// TIA Portal project "Project1" (V15.1)

(* hardware
DEVICE "S7-1200 station_1"  S7-1200 Station
   slot 0: "Rack_0"  S7-1200 Rack  Rack  V1.0
   slot 1: "PLC_1"  CPU 1214C AC/DC/Rly  6ES7 214-1BG40-0XB0  V4.2
DEVICE "HMI_1"  KTP700 Basic PN
   slot 0: "HMI_1"  KTP700 Basic PN  6AV2 123-2GB03-0AX0  15.1.0.0
   slot 1: "HMI_RT_1"  KTP700 Basic PN  6AV2 123-2GB03-0AX0  15.1.0.0
   slot 5: "HMI_1.IE_CP_1"  PROFINET Interface  15.0.1.0
      slot 1: "Interface PROFINET_1"  PROFINET Interface
         slot 1: "Port_1"  Port
*)

// ===== PLC "PLC_1"  CPU 1214C AC/DC/Rly =====

VAR_GLOBAL   // PLC tag table "Default tag table"
   "AU" AT %I0.0 : Bool;
   "X0" AT %M0.1 : Bool;
   "X30" AT %M0.2 : Bool;
   "Auto" AT %I0.3 : Bool;
   "Manuel" AT %I0.4 : Bool;
   "X31" AT %M0.5 : Bool;
   "X32" AT %M0.6 : Bool;
   "X20" AT %M0.7 : Bool;
   "BP1" AT %I1.0 : Bool;
   "BP2" AT %I1.2 : Bool;
   "X21" AT %M1.2 : Bool;
   "X22" AT %M1.4 : Bool;
   "CV1" AT %Q1.4 : Bool;
   "CV2" AT %Q1.6 : Bool;
   "NB1" AT %I1.6 : Bool;
   "NB2" AT %I1.7 : Bool;
   "X1" AT %M2.0 : Bool;
   "X2" AT %M2.1 : Bool;
   "X3" AT %M2.2 : Bool;
   "X4" AT %M2.3 : Bool;
   "X5" AT %M2.4 : Bool;
   "NH1" AT %I0.5 : Bool;
   "NH2" AT %I0.6 : Bool;
   "X10" AT %M2.7 : Bool;
   "X11" AT %M3.0 : Bool;
END_VAR

FUNCTION "GC" : Void   // FC1, LAD
{ S7_Optimized_Access := 'TRUE' }
VERSION : 0.1
BEGIN

REGION Network 1
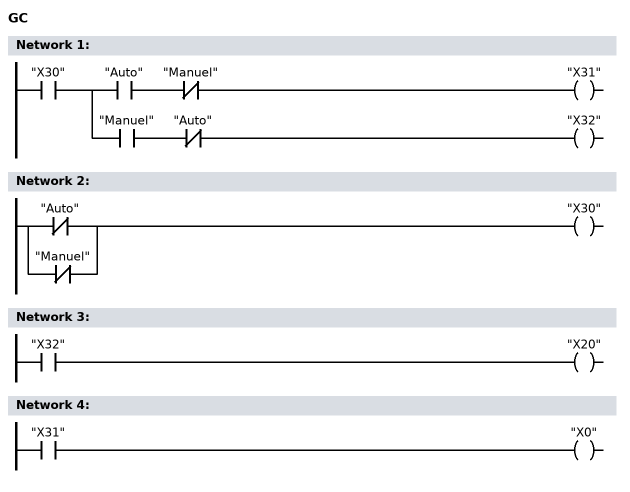
   RUNG wire#powerrail
      Contact( "X30" )
      wire#w1
      Contact( "Auto" )
      I_Contact( "Manuel" )
      Coil( "X31" )
   END_RUNG
   RUNG wire#w1
      Contact( "Manuel" )
      I_Contact( "Auto" )
      Coil( "X32" )
   END_RUNG
   // the same network as SCL:
   "X31" := "X30" AND "Auto" AND NOT "Manuel";
   "X32" := "X30" AND "Manuel" AND NOT "Auto";
END_REGION

REGION Network 2
   RUNG wire#powerrail
      I_Contact( "Auto" )
      wire#w1
      Coil( "X30" )
   END_RUNG
   RUNG wire#powerrail
      I_Contact( "Manuel" )
   END_RUNG wire#w1
   // the same network as SCL:
   "X30" := NOT "Auto" OR NOT "Manuel";
END_REGION

REGION Network 3
   RUNG wire#powerrail
      Contact( "X32" )
      Coil( "X20" )
   END_RUNG
   // the same network as SCL:
   "X20" := "X32";
END_REGION

REGION Network 4
   RUNG wire#powerrail
      Contact( "X31" )
      Coil( "X0" )
   END_RUNG
   // the same network as SCL:
   "X0" := "X31";
END_REGION
END_FUNCTION

FUNCTION "GMM" : Void   // FC2, LAD
{ S7_Optimized_Access := 'TRUE' }
VERSION : 0.1
   VAR_TEMP   // added for the SCL form of the ladder/FBD networks
      _w1 : Bool;
   END_VAR
BEGIN

REGION Network 1
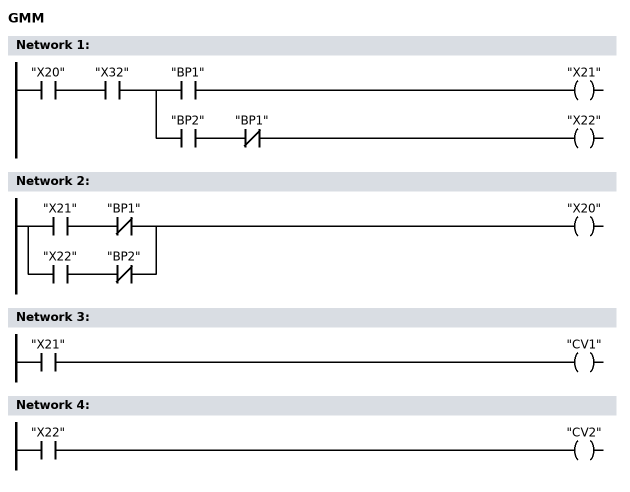
   RUNG wire#powerrail
      Contact( "X20" )
      Contact( "X32" )
      wire#w1
      Contact( "BP1" )
      Coil( "X21" )
   END_RUNG
   RUNG wire#w1
      Contact( "BP2" )
      I_Contact( "BP1" )
      Coil( "X22" )
   END_RUNG
   // the same network as SCL:
   #_w1 := "X20" AND "X32";
   "X21" := #_w1 AND "BP1";
   "X22" := #_w1 AND "BP2" AND NOT "BP1";
END_REGION

REGION Network 2
   RUNG wire#powerrail
      Contact( "X21" )
      I_Contact( "BP1" )
      wire#w1
      Coil( "X20" )
   END_RUNG
   RUNG wire#powerrail
      Contact( "X22" )
      I_Contact( "BP2" )
   END_RUNG wire#w1
   // the same network as SCL:
   "X20" := ("X21" AND NOT "BP1") OR ("X22" AND NOT "BP2");
END_REGION

REGION Network 3
   RUNG wire#powerrail
      Contact( "X21" )
      Coil( "CV1" )
   END_RUNG
   // the same network as SCL:
   "CV1" := "X21";
END_REGION

REGION Network 4
   RUNG wire#powerrail
      Contact( "X22" )
      Coil( "CV2" )
   END_RUNG
   // the same network as SCL:
   "CV2" := "X22";
END_REGION
END_FUNCTION

FUNCTION "GPN" : Void   // FC3, LAD
{ S7_Optimized_Access := 'TRUE' }
VERSION : 0.1
BEGIN

REGION Network 1
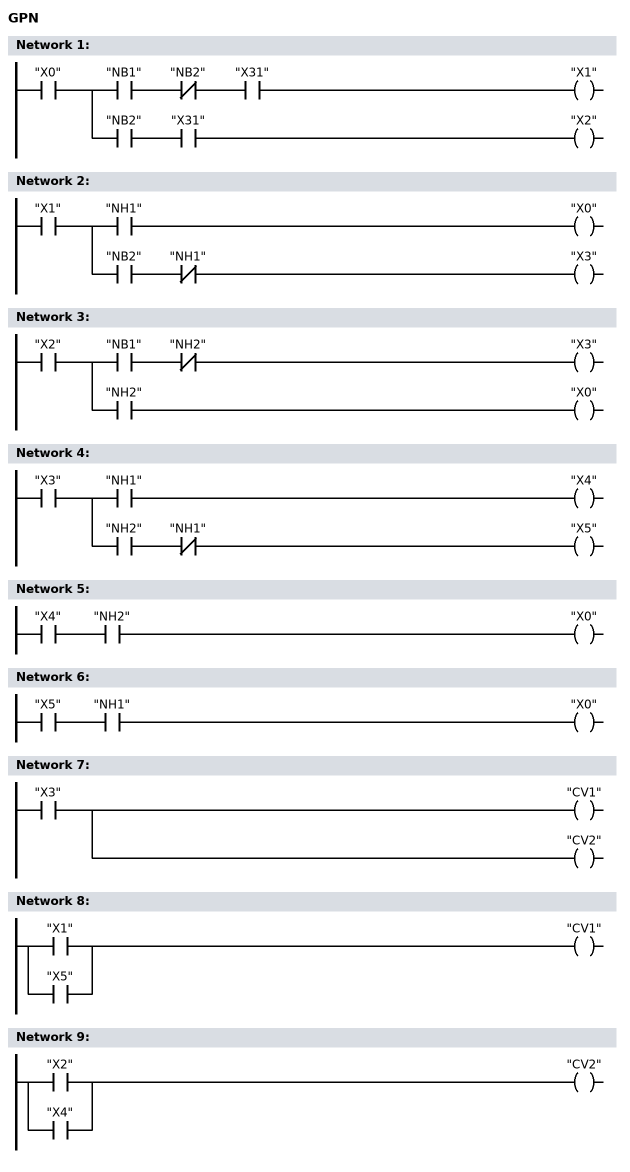
   RUNG wire#powerrail
      Contact( "X0" )
      wire#w1
      Contact( "NB1" )
      I_Contact( "NB2" )
      Contact( "X31" )
      Coil( "X1" )
   END_RUNG
   RUNG wire#w1
      Contact( "NB2" )
      Contact( "X31" )
      Coil( "X2" )
   END_RUNG
   // the same network as SCL:
   "X1" := "X0" AND "NB1" AND NOT "NB2" AND "X31";
   "X2" := "X0" AND "NB2" AND "X31";
END_REGION

REGION Network 2
   RUNG wire#powerrail
      Contact( "X1" )
      wire#w1
      Contact( "NH1" )
      Coil( "X0" )
   END_RUNG
   RUNG wire#w1
      Contact( "NB2" )
      I_Contact( "NH1" )
      Coil( "X3" )
   END_RUNG
   // the same network as SCL:
   "X0" := "X1" AND "NH1";
   "X3" := "X1" AND "NB2" AND NOT "NH1";
END_REGION

REGION Network 3
   RUNG wire#powerrail
      Contact( "X2" )
      wire#w1
      Contact( "NB1" )
      I_Contact( "NH2" )
      Coil( "X3" )
   END_RUNG
   RUNG wire#w1
      Contact( "NH2" )
      Coil( "X0" )
   END_RUNG
   // the same network as SCL:
   "X3" := "X2" AND "NB1" AND NOT "NH2";
   "X0" := "X2" AND "NH2";
END_REGION

REGION Network 4
   RUNG wire#powerrail
      Contact( "X3" )
      wire#w1
      Contact( "NH1" )
      Coil( "X4" )
   END_RUNG
   RUNG wire#w1
      Contact( "NH2" )
      I_Contact( "NH1" )
      Coil( "X5" )
   END_RUNG
   // the same network as SCL:
   "X4" := "X3" AND "NH1";
   "X5" := "X3" AND "NH2" AND NOT "NH1";
END_REGION

REGION Network 5
   RUNG wire#powerrail
      Contact( "X4" )
      Contact( "NH2" )
      Coil( "X0" )
   END_RUNG
   // the same network as SCL:
   "X0" := "X4" AND "NH2";
END_REGION

REGION Network 6
   RUNG wire#powerrail
      Contact( "X5" )
      Contact( "NH1" )
      Coil( "X0" )
   END_RUNG
   // the same network as SCL:
   "X0" := "X5" AND "NH1";
END_REGION

REGION Network 7
   RUNG wire#powerrail
      Contact( "X3" )
      wire#w1
      Coil( "CV1" )
   END_RUNG
   RUNG wire#w1
      Coil( "CV2" )
   END_RUNG
   // the same network as SCL:
   "CV1" := "X3";
   "CV2" := "X3";
END_REGION

REGION Network 8
   RUNG wire#powerrail
      Contact( "X1" )
      wire#w1
      Coil( "CV1" )
   END_RUNG
   RUNG wire#powerrail
      Contact( "X5" )
   END_RUNG wire#w1
   // the same network as SCL:
   "CV1" := "X1" OR "X5";
END_REGION

REGION Network 9
   RUNG wire#powerrail
      Contact( "X2" )
      wire#w1
      Coil( "CV2" )
   END_RUNG
   RUNG wire#powerrail
      Contact( "X4" )
   END_RUNG wire#w1
   // the same network as SCL:
   "CV2" := "X2" OR "X4";
END_REGION
END_FUNCTION

ORGANIZATION_BLOCK "Main"   // OB1, LAD, ProgramCycle
TITLE = "Main Program Sweep (Cycle)"
{ S7_Optimized_Access := 'TRUE' }
VERSION : 0.1
   VAR_INPUT
      Initial_Call : Bool;   // Initial call of this OB
      Remanence : Bool;   // =True, if remanent data are available
   END_VAR
   VAR_TEMP   // added for the SCL form of the ladder/FBD networks
      _w1 : Bool;
      _w2 : Bool;
   END_VAR
BEGIN

REGION Network 1
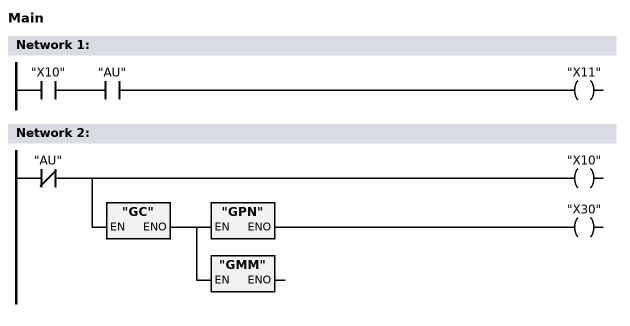
   RUNG wire#powerrail
      Contact( "X10" )
      Contact( "AU" )
      Coil( "X11" )
   END_RUNG
   // the same network as SCL:
   "X11" := "X10" AND "AU";
END_REGION

REGION Network 2
   RUNG wire#powerrail
      I_Contact( "AU" )
      wire#w1
      Coil( "X10" )
   END_RUNG
   RUNG wire#w1
      "GC"()
      wire#w2
      "GPN"()
      Coil( "X30" )
   END_RUNG
   RUNG wire#w2
      "GMM"()
   END_RUNG
   // the same network as SCL:
   "X10" := NOT "AU";
   "GC"(EN := NOT "AU", ENO => #_w1);
   "GPN"(EN := #_w1, ENO => #_w2);
   "X30" := #_w2;
   IF #_w1 THEN "GMM"(); END_IF;
END_REGION
END_ORGANIZATION_BLOCK

(* ===== HMI "HMI_RT_1" =====
system functions are stored by id; their names below are inferred from use
connection "HMI_Liaison_1": ETHERNET, SMART_S7_1200_OMS

HMI tags "Table de variables standard"
   "Numéro_vue_variable" : UInt, internal
   "NB1" : Bool = PLC NB1 AT %I1.6, 1 s
   "Auto" : Bool = PLC Auto AT %I0.3, 1 s

Template "Modèle_1" 800x480
   Button "Exit" at 714,429 size 71x50; TextOff 'Exit'; PictureOff "ExitRuntime_KTP700_Basic_PN_TR"; PictureOn "ExitRuntime_KTP700_Basic_PN_TR"
      on Release: StopRuntime(0)
   Button "Template_Button" at 614,429 size 71x50; TextOff 'Text'
   Button "Template_Button_1" at 514,429 size 71x50; TextOff 'Text'
   Button "Template_Button_2" at 414,429 size 71x50; TextOff 'Text'
   Button "Template_Button_3" at 314,429 size 71x50; TextOff 'Text'
   Button "Template_Button_4" at 214,429 size 71x50; TextOff 'Text'
   Button "Template_Button_5" at 114,429 size 71x50; TextOff 'Text'
   Button "Start screen" at 14,429 size 71x50; TextOff 'Start screen'; PictureOff "NavigateHome_KTP700_Basic_PN_TR"; PictureOn "NavigateHome_KTP700_Basic_PN_TR"
      on Release: ActivateScreen("Vue racine", 0)
   SymbolicIOField "Vue_champ_ES_symbolique" at 93,9 size 600x33; TextOff '0'; TextOn '1'; TextList "TextList_ScreenNames"
      ProcessValue <- "Numéro_vue_variable"
      on Change: ActivateScreenByNumber("Numéro_vue_variable", 0)
   DateTimeField "HmiScreenItemData" at 695,25 size 105x25
   DateTimeField "HmiScreenItemData_1" at 695,0 size 105x25
   GraphicView "Logo" at 0,0 size 91x51; Picture "Logo of HMI_1"

screen "Vue racine" 800x480, template "Modèle_1"
   on GenerateScreen: SetTag("Numéro_vue_variable", 1)
   TextField "HmiScreenItemData" at 80,225 size 640x25; Text 'Welcome to HMI_1 (KTP700 Basic+ PN)!'
   Ellipse "Ellipse_1" at 218,76 size 96x48
      Appearance <- "NB1"
   Button "Bouton_1" at 486,92 size 96x32; TextOff 'auto'
      Appearance <- "Auto"
      ProcessValue <- "Auto"
   Switch "Commutateur_1" at 427,158 size 64x32; CaptionText 'Switch'; TextOff 'manuel'; TextOn 'Auto'
      ProcessValue <- "Auto"
   SymbolicIOField "Champ d'E/S symbolique_1" at 191,150 size 96x32; TextOff '0'; TextOn '1'
      ProcessValue <- "Auto"
*)